ABB RobotStudio station: practica4.rspag

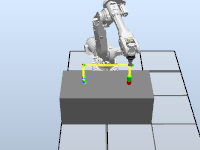
--- station ---
Station practica4 (saved by RobotStudio 20.4.9280.0)
Controller Controlador5
  mechanical unit ROB_1: IRB6640_180_255__04, 6 joints, base frame (0, 0, 0) mm
Layout (positions relative to the parent item):
  - Ventosa [mechanism] at (1500, 500, 1450) mm, rotated rx -180 ry 0 rz -180 deg
      TCP Ventosa at (0, 0, 200) mm
      links: PiezaVentosa
  - IRB6640_180_255__04 [mechanism, from Robots\IRB6640_180_255_G_04.rslib] at (0, 0, 0) mm; joint values [0.3218, 0.1103, 0.2349, 0, 1.2255, 0.3218] (rad or m)
  - Pieza_5 [part]
  - Pieza_6 [part]
  - Componente inteligente_1 [smart component]
      signals: DO PiezaDetectada, DO PiezaCogida, DI ActivaVentosa
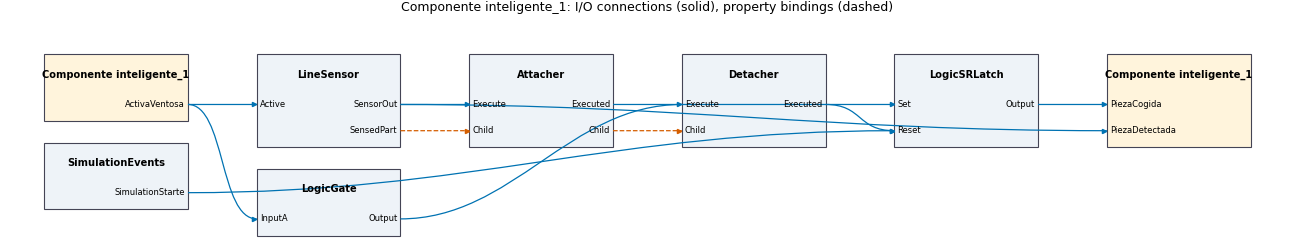
      connections:
        Componente inteligente_1.ActivaVentosa -> LineSensor.Active
        LineSensor.SensorOut -> Attacher.Execute
        Attacher.Executed -> LogicSRLatch.Set
        LogicSRLatch.Output -> Componente inteligente_1.PiezaCogida
        Componente inteligente_1.ActivaVentosa -> LogicGate.InputA
        LogicGate.Output -> Detacher.Execute
        Detacher.Executed -> LogicSRLatch.Reset
        SimulationEvents.SimulationStarted -> LogicSRLatch.Reset
        LineSensor.SensorOut -> Componente inteligente_1.PiezaDetectada
        LineSensor.SensedPart => Attacher.Child
        Attacher.Child => Detacher.Child
    - LineSensor [smart component, from Components\LineSensor.rslib] at (1500, 500, 1250) mm, rotated rx -180 ry 0 rz -180 deg
        properties: Start=[0 0 -0.002]; End=[0 0 0.02]; Radius=0.002; SensedPart=Pieza_8; SensedPoint=[1.5 0.5 0.95]
      - _sensorPart_ [part]
    - LogicSRLatch [smart component, from Components\LogicSRLatch.rslib]
    - SimulationEvents [smart component, from Components\SimulationEvents.rslib]
    - Attacher [smart component, from Components\Attacher.rslib]
        properties: Parent=Ventosa; Flange=0; Child=Pieza_8; Mount=false; Offset=[0 0 0]; Orientation=[0 0 0]
    - Detacher [smart component, from Components\Detacher.rslib]
        properties: Child=Pieza_8; KeepPosition=true
    - LogicGate [smart component, from Components\LogicGate.rslib]
        properties: Operator=NOT; Delay=0
  - Pieza_7 [part] at (0, 0, 0) mm
  - Pieza_8 [part] at (0, 0, 0) mm
Attachment: Ventosa is attached to IRB6640_180_255__04 / Link6
Attachment: LineSensor is attached to Ventosa / PiezaVentosa
Station logic (signal -> signal, property => property):
  Componente inteligente_1.PiezaDetectada -> Controlador5.ED_PiezaDetectada
  Controlador5.SD_ActivarVentosa -> Componente inteligente_1.ActivaVentosa
  Componente inteligente_1.PiezaCogida -> Controlador5.ED_PiezaCogida
Targets, tools, work objects and paths stored in the station and not in the controller backup, written as RAPID:
! task T_ROB1
MODULE Module1
  CONST robtarget pOrigenBase:=[[1500,500,750],[0,0,1,0],[0,0,0,0],[9E+09,9E+09,9E+09,9E+09,9E+09,9E+09]];
  CONST robtarget pDestinoBase:=[[1500,-500,750],[0,0,1,0],[0,0,0,0],[9E+09,9E+09,9E+09,9E+09,9E+09,9E+09]];
ENDMODULE


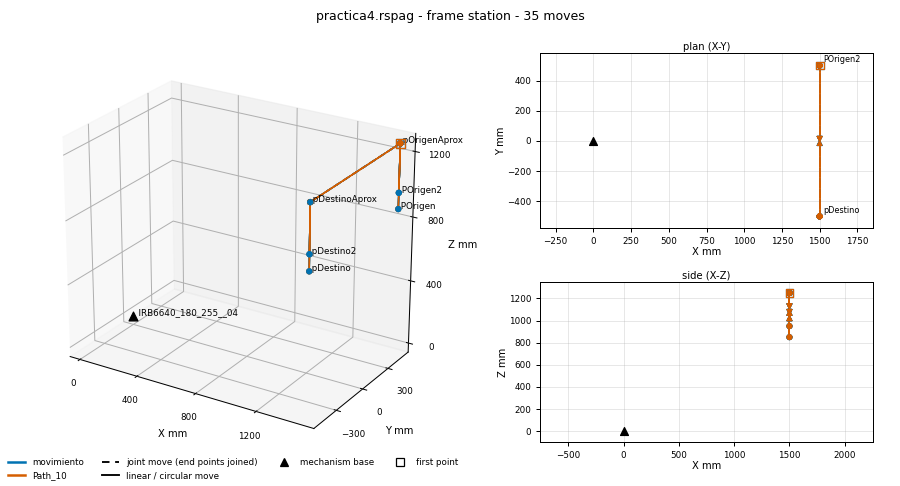
[picture p0: tool path of practica4.rspag in frame station, 35 of 35 moves have a stored position in this frame; points joined in program order, loops and branches not executed]
--- Backups/Controlador5/RAPID/TASK1/PROGMOD/CalibData.mod ---
MODULE CalibData
    PERS tooldata Ventosa:=[TRUE,[[0,0,200],[1,0,0,0]],[1,[0,0,125],[1,0,0,0],0.002,0.002,0.001]];
ENDMODULE

--- Backups/Controlador5/RAPID/TASK1/PROGMOD/Module1.mod ---
MODULE Module1
    CONST robtarget pOrigenAprox:=[[1499.999958379,499.999981236,1249.999954428],[0.000000004,0,1,0.000000001],[0,-1,0,0],[9E+09,9E+09,9E+09,9E+09,9E+09,9E+09]];
    CONST robtarget pOrigen:=[[1500,500,850],[0,0,1,0],[0,0,0,0],[9E+09,9E+09,9E+09,9E+09,9E+09,9E+09]];
    CONST robtarget pDestinoAprox:=[[1500,-500,1250],[0,0,1,0],[-1,0,-1,0],[9E+09,9E+09,9E+09,9E+09,9E+09,9E+09]];
    CONST robtarget pDestino:=[[1500,-500,850],[0,0,1,0],[-1,0,-1,0],[9E+09,9E+09,9E+09,9E+09,9E+09,9E+09]];
    CONST robtarget POrigen2:=[[1500,500,950],[0,0,1,0],[0,0,0,0],[9E+09,9E+09,9E+09,9E+09,9E+09,9E+09]];
    CONST robtarget pDestino2:=[[1500,-500,950],[0,0,1,0],[-1,0,-1,0],[9E+09,9E+09,9E+09,9E+09,9E+09,9E+09]];
!***********************************************************
    !
    ! Módulo:  Module1
    !
    ! Descripción:
    !   <Introduzca la descripción aquí>
    !
    ! Autor: franc
    !
    ! Versión: 1.0
    !
    !***********************************************************


    !***********************************************************
    !
    ! Procedimiento Main
    !
    !   Este es el punto de entrada de su programa
    !
    !***********************************************************
    PROC main()
        !Añada aquí su código
        movimiento;
    ENDPROC
    PROC movimiento()
        MoveJ pOrigenAprox,v2500,z100,Ventosa\WObj:=wobj0;
        MoveL POrigen2,v300,fine,Ventosa\WObj:=wobj0;
        SetDO SD_ActivarVentosa, 1; !Ponemos la ventosa a 1
        WaitDI ED_PiezaCogida, 1; !Esperamos a que PiezaCogida esté a 1, así no esperamos los dos segundos
        !WaitTime 2;
        MoveL pOrigenAprox,v300,z100,Ventosa\WObj:=wobj0;
        MoveJ pDestinoAprox,v2500,z100,Ventosa\WObj:=wobj0;
        MoveL pDestino,v300,fine,Ventosa\WObj:=wobj0;
        SetDO SD_ActivarVentosa, 0; !Ponemos la ventosa a 0, soltamos
        WaitDI ED_PiezaCogida, 0; !Esperamos a que PiezaCogida esté a 0, así no esperamos los dos segundos
        !WaitTime 2;
        MoveL pDestinoAprox,v300,z100,Ventosa\WObj:=wobj0;

        MoveJ pOrigenAprox,v2500,z100,Ventosa\WObj:=wobj0;
        MoveL POrigen,v300,fine,Ventosa\WObj:=wobj0;
        SetDO SD_ActivarVentosa, 1; !Ponemos la ventosa a 1
        WaitDI ED_PiezaCogida, 1; !Esperamos a que PiezaCogida esté a 1, así no esperamos los dos segundos
        !WaitTime 2;
        MoveL pOrigenAprox,v300,z100,Ventosa\WObj:=wobj0;
        MoveJ pDestinoAprox,v2500,z100,Ventosa\WObj:=wobj0;
        MoveL pDestino2,v300,fine,Ventosa\WObj:=wobj0;
        SetDO SD_ActivarVentosa, 0; !Ponemos la ventosa a 0, soltamos
        WaitDI ED_PiezaCogida, 0; !Esperamos a que PiezaCogida esté a 0, así no esperamos los dos segundos
        !WaitTime 2;
        MoveL pDestinoAprox,v300,z100,Ventosa\WObj:=wobj0;

        WaitTime 2;

        MoveL PDestino2,v300,fine,Ventosa\WObj:=wobj0;
        SetDO SD_ActivarVentosa, 1; !Ponemos la ventosa a 1
        WaitDI ED_PiezaCogida, 1; !Esperamos a que PiezaCogida esté a 1, así no esperamos los dos segundos
        !WaitTime 2;
        MoveL pDestinoAprox,v300,z100,Ventosa\WObj:=wobj0;
        MoveJ pOrigenAprox,v2500,z100,Ventosa\WObj:=wobj0;
        MoveL pOrigen,v300,fine,Ventosa\WObj:=wobj0;
        SetDO SD_ActivarVentosa, 0; !Ponemos la ventosa a 0, soltamos
        WaitDI ED_PiezaCogida, 0; !Esperamos a que PiezaCogida esté a 0, así no esperamos los dos segundos
        !WaitTime 2;
        MoveL pOrigenAprox,v300,z100,Ventosa\WObj:=wobj0;

        MoveJ pDestinoAprox,v2500,z100,Ventosa\WObj:=wobj0;
        MoveL PDestino,v300,fine,Ventosa\WObj:=wobj0;
        SetDO SD_ActivarVentosa, 1; !Ponemos la ventosa a 1
        WaitDI ED_PiezaCogida, 1; !Esperamos a que PiezaCogida esté a 1, así no esperamos los dos segundos
        !WaitTime 2;
        MoveL pDestinoAprox,v300,z100,Ventosa\WObj:=wobj0;
        MoveJ pOrigenAprox,v2500,z100,Ventosa\WObj:=wobj0;
        MoveL pOrigen2,v300,fine,Ventosa\WObj:=wobj0;
        SetDO SD_ActivarVentosa, 0; !Ponemos la ventosa a 0, soltamos
        WaitDI ED_PiezaCogida, 0; !Esperamos a que PiezaCogida esté a 0, así no esperamos los dos segundos
        !WaitTime 2;
        MoveL pOrigenAprox,v300,z100,Ventosa\WObj:=wobj0;


    ENDPROC
    PROC Path_10()
        MoveJ pOrigenAprox,v2500,z100,Ventosa\WObj:=wobj0;
        MoveL POrigen2,v1000,fine,Ventosa\WObj:=wobj0;
        MoveL pOrigenAprox,v300,z100,Ventosa\WObj:=wobj0;
        MoveJ pDestinoAprox,v2500,z100,Ventosa\WObj:=wobj0;
        MoveL pDestino,v300,fine,Ventosa\WObj:=wobj0;
        MoveL pDestinoAprox,v300,z100,Ventosa\WObj:=wobj0;
        MoveL pOrigenAprox,v1000,z100,Ventosa\WObj:=wobj0;
        MoveL pOrigen,v1000,z100,Ventosa\WObj:=wobj0;
        MoveL pOrigenAprox,v1000,z100,Ventosa\WObj:=wobj0;
        MoveL pDestinoAprox,v1000,z100,Ventosa\WObj:=wobj0;
        MoveL pDestino2,v1000,fine,Ventosa\WObj:=wobj0;
        MoveL pDestinoAprox,v1000,z100,Ventosa\WObj:=wobj0;
    ENDPROC
ENDMODULE

--- Backups/Controlador5/SYSPAR/EIO.cfg ---
EIO:CFG_1.0:6:1::
#
INDUSTRIAL_NETWORK:

      -Name "DeviceNet" -Label "DeviceNet Master/Slave Network" -Address "2"
#
DEVICENET_DEVICE:

      -Name "MiDeviceNet"
#
DEVICENET_INTERNAL_DEVICE:

      -Name "DN_Internal_Device" -VendorName "ABB Robotics"\
      -ProductName "DeviceNet Internal Slave Device"
#
EIO_SIGNAL:

      -Name "ED_PiezaDetectada" -SignalType "DI" -Device "MiDeviceNet"\
      -Label "ED_PiezaDetectada" -DeviceMap "0" -Access "All"

      -Name "ED_PiezaCogida" -SignalType "DI" -Device "MiDeviceNet"\
      -Label "ED_PiezaCogida" -DeviceMap "1" -Access "All"

      -Name "SD_ActivarVentosa" -SignalType "DO" -Device "MiDeviceNet"\
      -Label "SD_ActivarVentosa" -DeviceMap "0" -Access "All"
